Staubli VAL3: OnF1.pgx

program OnF1()
begin
  switch nPage
    case 0
      call Edit(sItem)
    break
    case 1
      switch nSelected
        case 0
          uPallet[sItem].pO=here(tTool,world)
          popUpMsg("OK")
        break
        case 1
          uPallet[sItem].pO=here(tTool,world)
          popUpMsg("OK")
        break
        case 2
          uPallet[sItem].pO=here(tTool,world)
          popUpMsg("OK")
        break
      endSwitch
    break

  endSwitch
end
